(* PLC project Unnamed, Unknown Unnamed 1 *)
(* stored: creationDateTime 2024-11-03T12:34:03, modificationDateTime 2024-11-06T21:45:40 *)

PROGRAM program0
  VAR
    Traffic_A : BOOL;
    Traffic_B : BOOL;
    AtoB_Amber : BOOL;
    BtoA_Amber : BOOL;
    A_Crossing_A_Amber : BOOL;
    A_Crossing_B_Amber : BOOL;
    B_Crossing_A_Amber : BOOL;
    B_Crossing_B_Amber : BOOL;
    A_Crossing_A : BOOL;
    A_Crossing_B : BOOL;
    B_Crossing_A : BOOL;
    B_Crossing_B : BOOL;
  END_VAR
  VAR
    Change AT %IX0.5 : BOOL;
    Cross_A AT %IX0.6 : BOOL;
    Cross_B AT %IX0.7 : BOOL;
  END_VAR
  VAR
    Amber_Dwell : TIME := T#2s;
    Crossing_Dwell : TIME := T#3s;
    Traffic_Dwell : TIME := T#5s;
    TON0 : TON;
    TON1 : TON;
    TON2 : TON;
    TON3 : TON;
    TON4 : TON;
    TON5 : TON;
    TON6 : TON;
    TON7 : TON;
    TON8 : TON;
  END_VAR
  VAR
    Red_B AT %QX0.5 : BOOL;
    Amber_B AT %QX0.4 : BOOL;
    Green_B AT %QX0.3 : BOOL;
    Stop_B AT %QX0.7 : BOOL;
    Red_A AT %QX0.2 : BOOL;
    Amber_A AT %QX0.1 : BOOL;
    Green_A AT %QX0.0 : BOOL;
    Stop_A AT %QX0.6 : BOOL;
  END_VAR
  VAR
    Crossing_A_Latch : BOOL;
    Crossing_B_Latch : BOOL;
    TON9 : TON;
    TON10 : TON;
    TON11 : TON;
    TON12 : TON;
  END_VAR

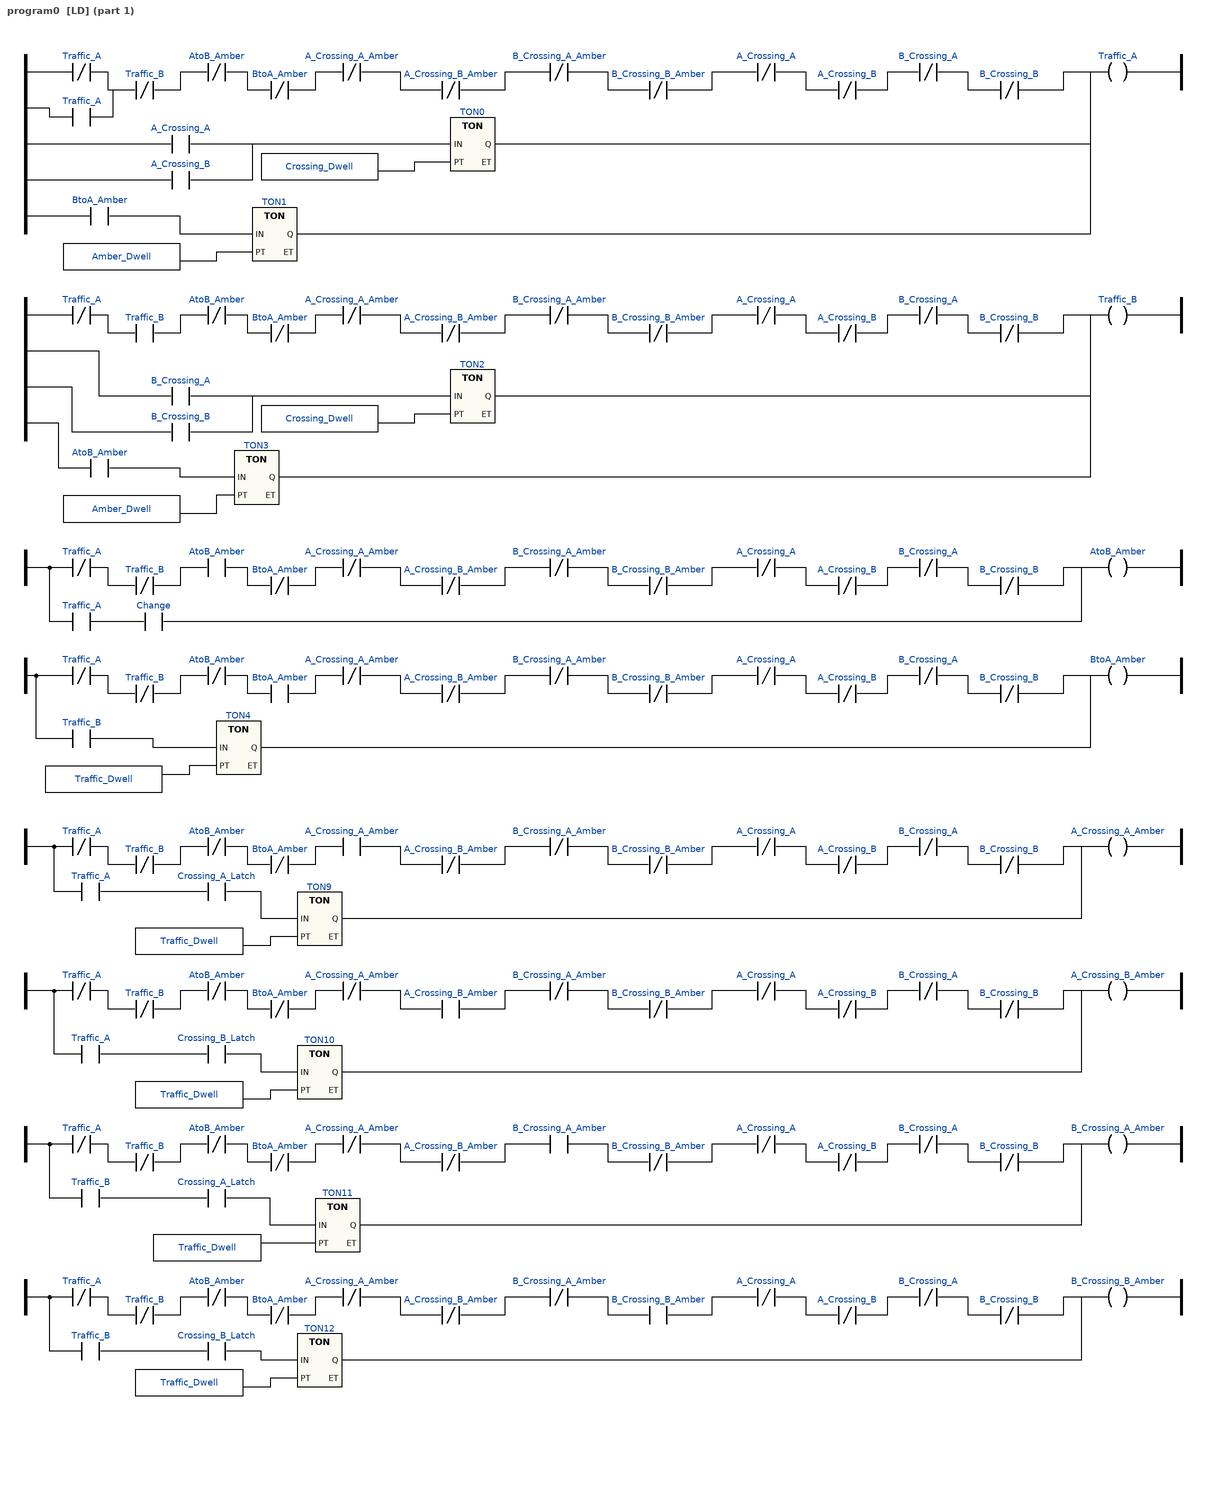
(* LD diagram, written out as Structured Text *)
TON1(IN := BtoA_Amber, PT := Amber_Dwell);
TON0(IN := A_Crossing_B OR A_Crossing_A, PT := Crossing_Dwell);
Traffic_A := (NOT Traffic_A OR Traffic_A) AND NOT Traffic_B AND NOT AtoB_Amber AND NOT BtoA_Amber AND NOT A_Crossing_A_Amber AND NOT A_Crossing_B_Amber AND NOT B_Crossing_A_Amber AND NOT B_Crossing_B_Amber AND NOT A_Crossing_A AND NOT A_Crossing_B AND NOT B_Crossing_A AND NOT B_Crossing_B OR TON1.Q OR TON0.Q;
TON2(IN := B_Crossing_B OR B_Crossing_A, PT := Crossing_Dwell);
TON3(IN := AtoB_Amber, PT := Amber_Dwell);
Traffic_B := NOT Traffic_A AND Traffic_B AND NOT AtoB_Amber AND NOT BtoA_Amber AND NOT A_Crossing_A_Amber AND NOT A_Crossing_B_Amber AND NOT B_Crossing_A_Amber AND NOT B_Crossing_B_Amber AND NOT A_Crossing_A AND NOT A_Crossing_B AND NOT B_Crossing_A AND NOT B_Crossing_B OR TON2.Q OR TON3.Q;
AtoB_Amber := NOT Traffic_A AND NOT Traffic_B AND AtoB_Amber AND NOT BtoA_Amber AND NOT A_Crossing_A_Amber AND NOT A_Crossing_B_Amber AND NOT B_Crossing_A_Amber AND NOT B_Crossing_B_Amber AND NOT A_Crossing_A AND NOT A_Crossing_B AND NOT B_Crossing_A AND NOT B_Crossing_B OR Traffic_A AND Change;
TON4(IN := Traffic_B, PT := Traffic_Dwell);
BtoA_Amber := NOT Traffic_A AND NOT Traffic_B AND NOT AtoB_Amber AND BtoA_Amber AND NOT A_Crossing_A_Amber AND NOT A_Crossing_B_Amber AND NOT B_Crossing_A_Amber AND NOT B_Crossing_B_Amber AND NOT A_Crossing_A AND NOT A_Crossing_B AND NOT B_Crossing_A AND NOT B_Crossing_B OR TON4.Q;
TON9(IN := Traffic_A AND Crossing_A_Latch, PT := Traffic_Dwell);
A_Crossing_A_Amber := NOT Traffic_A AND NOT Traffic_B AND NOT AtoB_Amber AND NOT BtoA_Amber AND A_Crossing_A_Amber AND NOT A_Crossing_B_Amber AND NOT B_Crossing_A_Amber AND NOT B_Crossing_B_Amber AND NOT A_Crossing_A AND NOT A_Crossing_B AND NOT B_Crossing_A AND NOT B_Crossing_B OR TON9.Q;
TON10(IN := Traffic_A AND Crossing_B_Latch, PT := Traffic_Dwell);
A_Crossing_B_Amber := NOT Traffic_A AND NOT Traffic_B AND NOT AtoB_Amber AND NOT BtoA_Amber AND NOT A_Crossing_A_Amber AND A_Crossing_B_Amber AND NOT B_Crossing_A_Amber AND NOT B_Crossing_B_Amber AND NOT A_Crossing_A AND NOT A_Crossing_B AND NOT B_Crossing_A AND NOT B_Crossing_B OR TON10.Q;
TON11(IN := Traffic_B AND Crossing_A_Latch, PT := Traffic_Dwell);
B_Crossing_A_Amber := NOT Traffic_A AND NOT Traffic_B AND NOT AtoB_Amber AND NOT BtoA_Amber AND NOT A_Crossing_A_Amber AND NOT A_Crossing_B_Amber AND B_Crossing_A_Amber AND NOT B_Crossing_B_Amber AND NOT A_Crossing_A AND NOT A_Crossing_B AND NOT B_Crossing_A AND NOT B_Crossing_B OR TON11.Q;
TON12(IN := Traffic_B AND Crossing_B_Latch, PT := Traffic_Dwell);
B_Crossing_B_Amber := NOT Traffic_A AND NOT Traffic_B AND NOT AtoB_Amber AND NOT BtoA_Amber AND NOT A_Crossing_A_Amber AND NOT A_Crossing_B_Amber AND NOT B_Crossing_A_Amber AND B_Crossing_B_Amber AND NOT A_Crossing_A AND NOT A_Crossing_B AND NOT B_Crossing_A AND NOT B_Crossing_B OR TON12.Q;
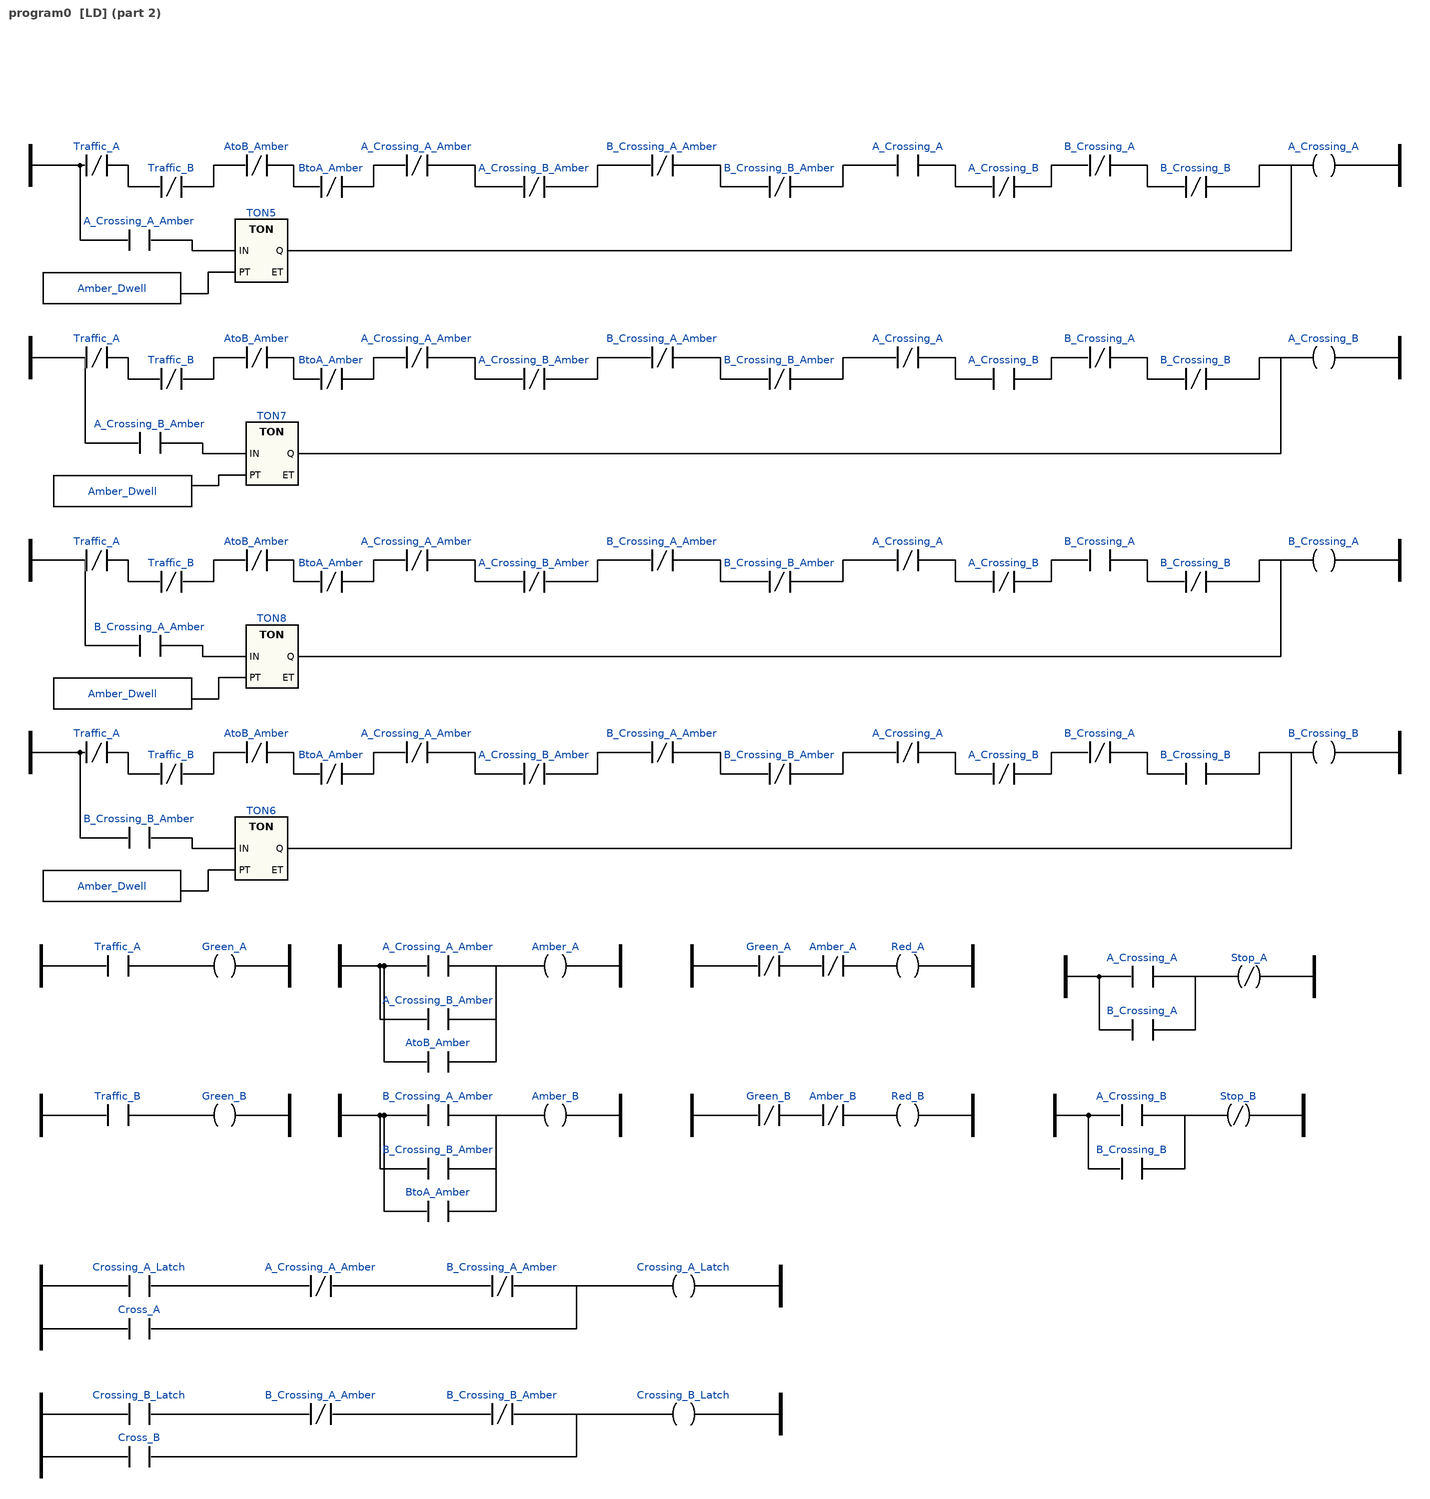
TON5(IN := A_Crossing_A_Amber, PT := Amber_Dwell);
A_Crossing_A := NOT Traffic_A AND NOT Traffic_B AND NOT AtoB_Amber AND NOT BtoA_Amber AND NOT A_Crossing_A_Amber AND NOT A_Crossing_B_Amber AND NOT B_Crossing_A_Amber AND NOT B_Crossing_B_Amber AND A_Crossing_A AND NOT A_Crossing_B AND NOT B_Crossing_A AND NOT B_Crossing_B OR TON5.Q;
TON7(IN := A_Crossing_B_Amber, PT := Amber_Dwell);
A_Crossing_B := NOT Traffic_A AND NOT Traffic_B AND NOT AtoB_Amber AND NOT BtoA_Amber AND NOT A_Crossing_A_Amber AND NOT A_Crossing_B_Amber AND NOT B_Crossing_A_Amber AND NOT B_Crossing_B_Amber AND NOT A_Crossing_A AND A_Crossing_B AND NOT B_Crossing_A AND NOT B_Crossing_B OR TON7.Q;
TON8(IN := B_Crossing_A_Amber, PT := Amber_Dwell);
B_Crossing_A := NOT Traffic_A AND NOT Traffic_B AND NOT AtoB_Amber AND NOT BtoA_Amber AND NOT A_Crossing_A_Amber AND NOT A_Crossing_B_Amber AND NOT B_Crossing_A_Amber AND NOT B_Crossing_B_Amber AND NOT A_Crossing_A AND NOT A_Crossing_B AND B_Crossing_A AND NOT B_Crossing_B OR TON8.Q;
TON6(IN := B_Crossing_B_Amber, PT := Amber_Dwell);
B_Crossing_B := NOT Traffic_A AND NOT Traffic_B AND NOT AtoB_Amber AND NOT BtoA_Amber AND NOT A_Crossing_A_Amber AND NOT A_Crossing_B_Amber AND NOT B_Crossing_A_Amber AND NOT B_Crossing_B_Amber AND NOT A_Crossing_A AND NOT A_Crossing_B AND NOT B_Crossing_A AND B_Crossing_B OR TON6.Q;
Green_A := Traffic_A;
Amber_A := A_Crossing_A_Amber OR AtoB_Amber OR A_Crossing_B_Amber;
Red_A := NOT Green_A AND NOT Amber_A;
Green_B := Traffic_B;
Amber_B := B_Crossing_A_Amber OR BtoA_Amber OR B_Crossing_B_Amber;
Red_B := NOT Green_B AND NOT Amber_B;
Stop_A := NOT (A_Crossing_A OR B_Crossing_A);
Stop_B := NOT (A_Crossing_B OR B_Crossing_B);
Crossing_A_Latch := Cross_A OR Crossing_A_Latch AND NOT A_Crossing_A_Amber AND NOT B_Crossing_A_Amber;
Crossing_B_Latch := Cross_B OR Crossing_B_Latch AND NOT B_Crossing_A_Amber AND NOT B_Crossing_B_Amber;
END_PROGRAM

CONFIGURATION Config0
  RESOURCE Res0 ON PLC
    TASK task0(INTERVAL := T#50ms, PRIORITY := 0);
    PROGRAM instance0 WITH task0 : program0;
  END_RESOURCE
END_CONFIGURATION
